(****************************************************************************************)
(*							Beckhoff Automation Poland									*)
(*								L_TBSquareWave v1.0										*)
(*									29.02.2007											*)
(*	This FB can be used to generate a Boolean square wave signal with a variable high/low time *)
(*______________________________________________________________________________________*)
FUNCTION_BLOCK L_TBSquareWave
VAR_INPUT
	bEnable:BOOL;
	wTimeHigh:WORD;
	wTimeLow:WORD;
END_VAR
VAR_OUTPUT
	bOut:BOOL;
END_VAR
VAR
	ton1: TON;
	ton2: TON;
END_VAR

IF bEnable THEN
	ton1(IN:= NOT ton2.Q, PT:=WORD_TO_TIME(wTimeLow));
	bOut:=NOT ton1.Q;
	ton2(IN:=ton1.Q , PT:=WORD_TO_TIME(wTimeHigh));
ELSE
	bOut:=FALSE;
END_IF

END_FUNCTION_BLOCK

(* stored: Version 1.1.0.1, ProductVersion 3.1.4026.13, FileIdentifier 9c041b44356e467794499c9d2bdaf2ecf845ac2c, FileSignature 0995ee491c181b00e3456ebd6a9b9d9f5a1219658763b1dd6f67cb542d0e68c1eae9772e4012efce164e947b054f3313776dc38f0f518c73da67ac94948f9bab82285501a833b8eff81d4e4ed8aa79a8de2b25d3b3b197dd5308ef46c46e13a1c411d84f88e495a79d2db4e1c1851977650458550239cc34aaadd942e21d18d25160c9aa39338b9976f8f62f541dfffbb9dc12305cf60a53d6345060881ba879ce79570390af6fae2125f197fba57ed29f773edc07b9bd01097218206433d913e3c9f1449dad934ea62d880add1544c231c978c500ab69b87f0dc98a038b4af919fc23bdddaa35b5f3b68c3b7617340e3032755ab8d279ec9ef3af26106230a4
   POU L_TBSquareWave: Id {a62201e8-5e33-4d17-865c-94d74d6a0145}, SpecialFunc None *)
